RoboDK station: PRUEBA_CIRCULO.rdk

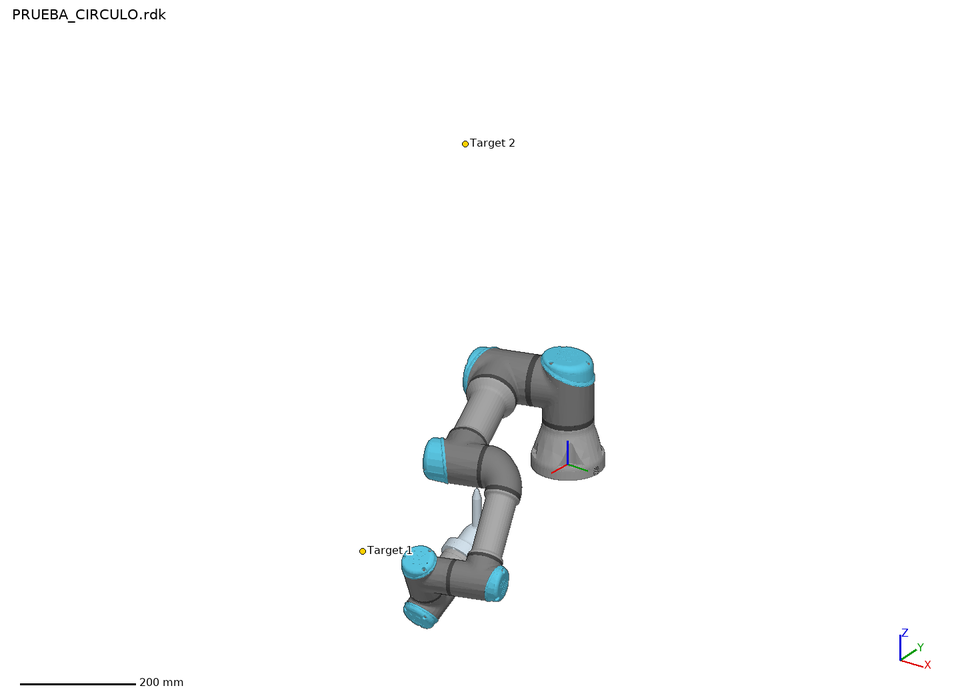
[picture v0: the station drawn from its stored meshes, robots at their saved joint values, targets as dots, program paths as lines]
Station PRUEBA_CIRCULO (saved by RoboDK 6.0.1). Poses are relative to the parent item; angles as X-Y-Z fixed-axis rotations.
  - frame UR3e Base at (-1.58, -22.27, 0) mm, rotated rx 0 ry -0.02 rz -94.05 deg
    - robot UR3e: 6 axes, payload 3 kg, reach 500 mm, repeatability 0.03 mm, weight 11 kg
        modified DH rows (alpha deg, a mm, theta deg, d mm): 0, 0, 0, 151.9; 90, 0, 180, 0; 0, 243.55, 0, 0; 0, 213.2, 0, 131.05; -90, 0, 0, 85.35; 90, 0, 180, 92.1
        joint limits [-360, -360, -360, -360, -360, -360] to [360, 360, 360, 360, 360, 360]; home [0, -90, -90, 0, 90, 0]; saved at [20.352, -193.833, -26.9, 189.108, 107.529, 79.493]
      - tool Generic Pencil Tool, TCP at (82.2, 0, 101.78) mm, rotated rx 0 ry 60 rz 0 deg, size 125 x 74.9 x 107.3 mm
    - target Target 1 (Cartesian target) at (538.68, -19.79, 30.04) mm, rotated rx 180 ry -1.36 rz 180 deg; joints [158.931, -33.367, -279.535, 166.054, -72.124, 78.662] of UR3e
    - target Target 2 (Cartesian target) at (280.37, 0, 721.78) mm, rotated rx 0 ry 81.99 rz 0 deg; joints [94.977, -118.182, 39.307, 350.881, 68.095, -5.365] of UR3e
    - frame Frame 1 at (0, 0.06, 0) mm
  - Python program Prog1 (listed below)
  - program Prog2 (3 instructions, listed below)

--- Python program Prog1 ---
# -*- coding: utf-8 -*-
from robodk.robolink import *
from robodk.robomath import *
import math

RDK = Robolink()
RDK.setRunMode(RUNMODE_SIMULATE)

# ----------- PARÁMETROS -----------
RADIO_MM        = 50.0
ALTURA_Z        = 15.0      # altura final del lápiz respecto a la base
PUNTOS          = 36        # 1 punto cada 10°

# ----------- OBJETOS -----------
robot = RDK.Item('', ITEM_TYPE_ROBOT)
base  = RDK.Item('UR3e Base', ITEM_TYPE_FRAME)
tool  = robot.getLink(ITEM_TYPE_TOOL)
t1    = RDK.Item('Target 1', ITEM_TYPE_TARGET)

robot.setFrame(base)
robot.setTool(tool)

# Pose del centro del círculo: Target 1
pose_center = t1.Pose()
xc, yc, _ = pose_center.Pos()

# ----------- GENERAR PUNTOS DEL CÍRCULO -----------
pts = []
for i in range(PUNTOS):
    ang = math.radians(i * (360.0 / PUNTOS))
    x = xc + RADIO_MM * math.cos(ang)
    y = yc + RADIO_MM * math.sin(ang)
    p = pose_center.copy()
    p.setPos([x, y, ALTURA_Z])
    pts.append(p)

try:
    # 1) Ir a Target 1 (posición inicial)
    robot.MoveJ(t1)

    # 2) Bajar el lápiz verticalmente hasta Z=15 mm
    px, py, _ = pose_center.Pos()
    p_down = pose_center.copy()
    p_down.setPos([px, py, ALTURA_Z])
    robot.MoveL(p_down)

    # 3) Dibujar círculo punto a punto
    for p in pts:
        robot.MoveL(p)

    # 4) Subir en vertical 30 mm
    p_up = pose_center.copy()
    p_up.setPos([px, py, ALTURA_Z + 30])
    robot.MoveL(p_up)

    # 5) Volver a target 1
    robot.MoveJ(t1)

    print("✔ Círculo completado correctamente.")

except Exception as e:
    print("Error:", e)

--- program Prog2 (robot UR3e) ---
  Est. Ref.: UR3e Base
  Est. herr: Generic Pencil Tool
  MoveJ (Target 2)
